# EPICS StreamDevice protocol: Pfeiffer/TPG256A.proto
## https://epics.anl.gov/tech-talk/2021/msg00373.php ##
## https://gitlab.esss.lu.se/epics-modules/vac/vac_ctrl_tpg300_500 ##

#################################################
# ###                                       ### #
# ### StreamDevice Protocol for             ### #
# ### Pfeiffer TPG256A                      ### #
# ###                                       ### #
# ### author: F.Feldbauer                   ### #
# ###                                       ### #
# ### Ref 1.0; 2011-05-19                   ### #
#################################################

###################
# ### Globals ### #
###################
#Terminator    = '';
OutTerminator = LF;
InTerminator = CR LF;
LockTimeout   = 5000;
ReplyTimeout  = 4000;
ReadTimeout   = 500;
WriteTimeout  = 3000;
ExtraInput    = Ignore;

##############################
# ### Exception Handlers ### #
##############################

#####################
# ### Protocols ### #
#####################
readout {
  out "PRX";
  in  ACK;
  out ENQ;
  in "%i,%E";
  # in  "%(\$2.VAL)i,%E\r\n";
  #in  "%(\$2.VAL)i,%E";
}
